// Mitsubishi GX Developer project: PLC_PCO520L2   PLC: Q06UDEH   RS485 Communication_STX

PROGRAM ST340_RS
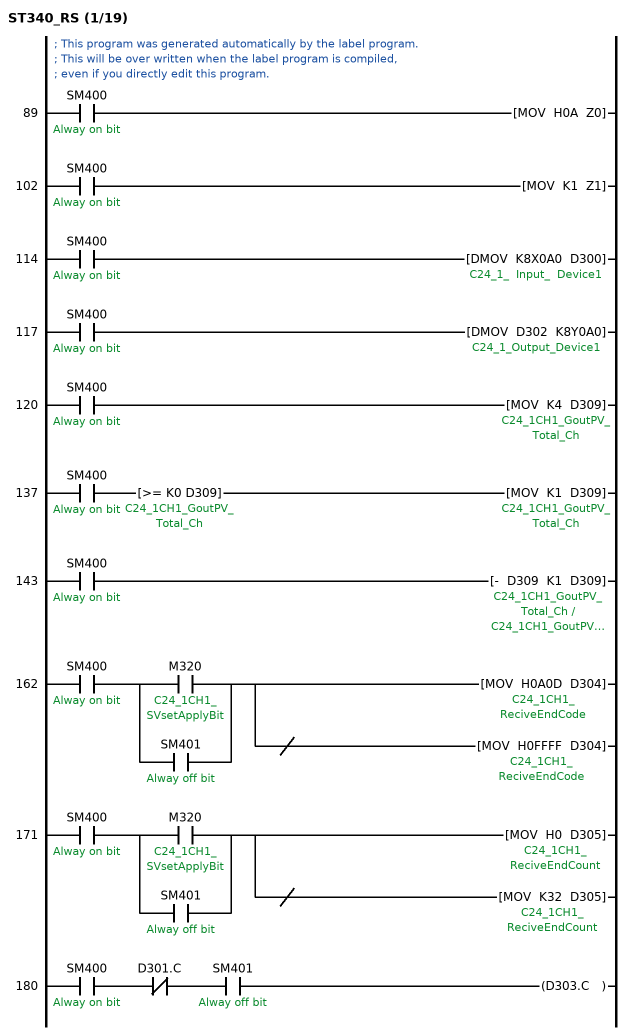
; This program was generated automatically by the label program.
; This will be over written when the label program is compiled,
; even if you directly edit this program.
89    LD      SM400  ; Alway on bit
      MOV     H0A Z0
        [note] Module IO Number
102   LD      SM400  ; Alway on bit
      MOV     K1 Z1
        [note] Channel Number
114   LD      SM400  ; Alway on bit
      DMOV    K8X0A0 D300  ; CH1 Transmission normal completi / C24_1_  Input_  Device1
117   LD      SM400  ; Alway on bit
      DMOV    D302 K8Y0A0  ; C24_1_Output_Device1 / CH1 Transmission request
120   LD      SM400  ; Alway on bit
      MOV     K4 D309  ; C24_1CH1_GoutPV_Total_Ch
        [note] Controller Channel Count
137   LD      SM400  ; Alway on bit
      AND>=   K0 D309  ; C24_1CH1_GoutPV_Total_Ch
      MOV     K1 D309
143   LD      SM400  ; Alway on bit
      -       D309 K1 D309
        [note] Controller Channel Count
162   LD      SM400  ; Alway on bit
      LD      M320  ; C24_1CH1_SVsetApplyBit
      OR      SM401  ; Alway off bit
      ANB
      MOV     H0A0D D304  ; C24_1CH1_ReciveEndCode
      INV
      MOV     H0FFFF D304
171   LD      SM400  ; Alway on bit
      LD      M320  ; C24_1CH1_SVsetApplyBit
      OR      SM401  ; Alway off bit
      ANB
      MOV     H0 D305  ; C24_1CH1_ReciveEndCount
      INV
      MOV     K32 D305
180   LD      SM400  ; Alway on bit
      ANI     D301.C
      AND     SM401  ; Alway off bit
      OUT     D303.C
        [note] System汲沥檬扁拳
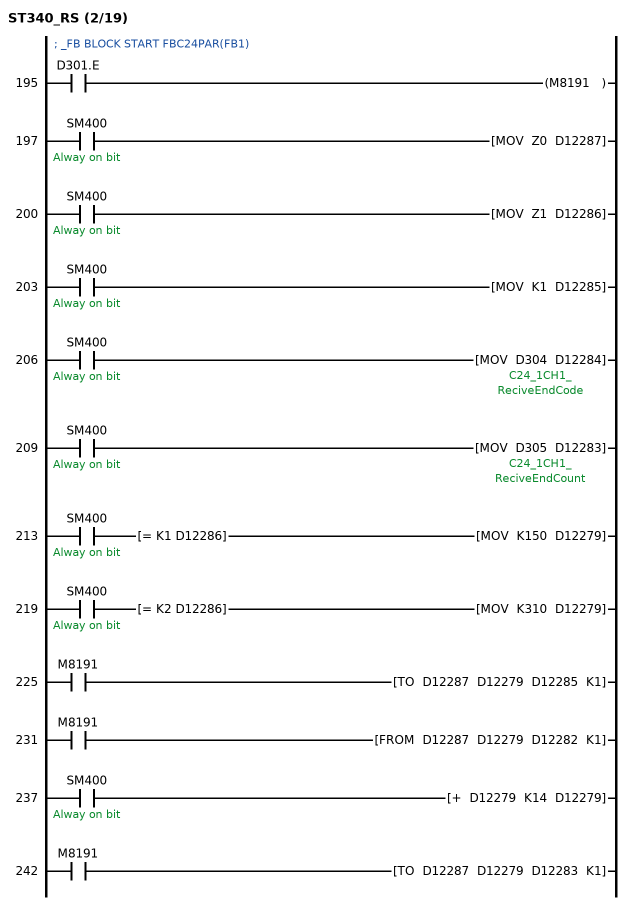
; _FB BLOCK START FBC24PAR(FB1)
195   LD      D301.E
      OUT     M8191
197   LD      SM400  ; Alway on bit
      MOV     Z0 D12287
200   LD      SM400  ; Alway on bit
      MOV     Z1 D12286
203   LD      SM400  ; Alway on bit
      MOV     K1 D12285
206   LD      SM400  ; Alway on bit
      MOV     D304 D12284
209   LD      SM400  ; Alway on bit
      MOV     D305 D12283
; FB START
213   LD      SM400  ; Alway on bit
      AND=    K1 D12286
      MOV     K150 D12279
219   LD      SM400  ; Alway on bit
      AND=    K2 D12286
      MOV     K310 D12279
225   LD      M8191
      TO      D12287 D12279 D12285 K1
231   LD      M8191
      FROM    D12287 D12279 D12282 K1
237   LD      SM400  ; Alway on bit
      +       D12279 K14 D12279
242   LD      M8191
      TO      D12287 D12279 D12283 K1
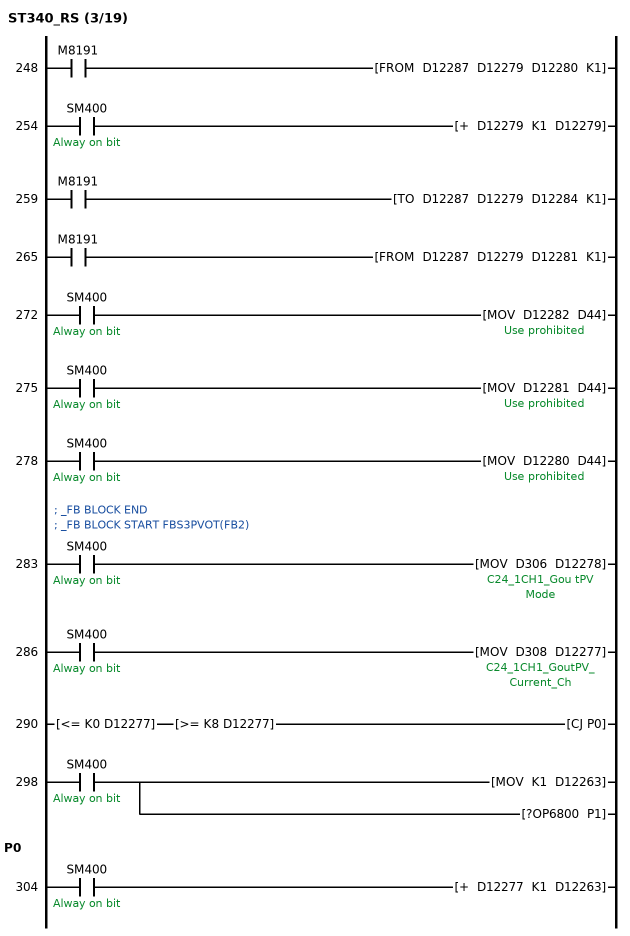
248   LD      M8191
      FROM    D12287 D12279 D12280 K1
254   LD      SM400  ; Alway on bit
      +       D12279 K1 D12279
259   LD      M8191
      TO      D12287 D12279 D12284 K1
265   LD      M8191
      FROM    D12287 D12279 D12281 K1
; FB END
272   LD      SM400  ; Alway on bit
      MOV     D12282 D44  ; Use prohibited
275   LD      SM400  ; Alway on bit
      MOV     D12281 D44
278   LD      SM400  ; Alway on bit
      MOV     D12280 D44
; _FB BLOCK END
; _FB BLOCK START FBS3PVOT(FB2)
283   LD      SM400  ; Alway on bit
      MOV     D306 D12278  ; C24_1CH1_Gou tPV Mode
286   LD      SM400  ; Alway on bit
      MOV     D308 D12277  ; C24_1CH1_GoutPV_Current_Ch
; FB START
290   LD<=    K0 D12277
      AND>=   K8 D12277
      CJ      P0
298   LD      SM400  ; Alway on bit
      MOV     K1 D12263
      ?OP6800 P1
      P0
304   LD      SM400  ; Alway on bit
      +       D12277 K1 D12263
      P1
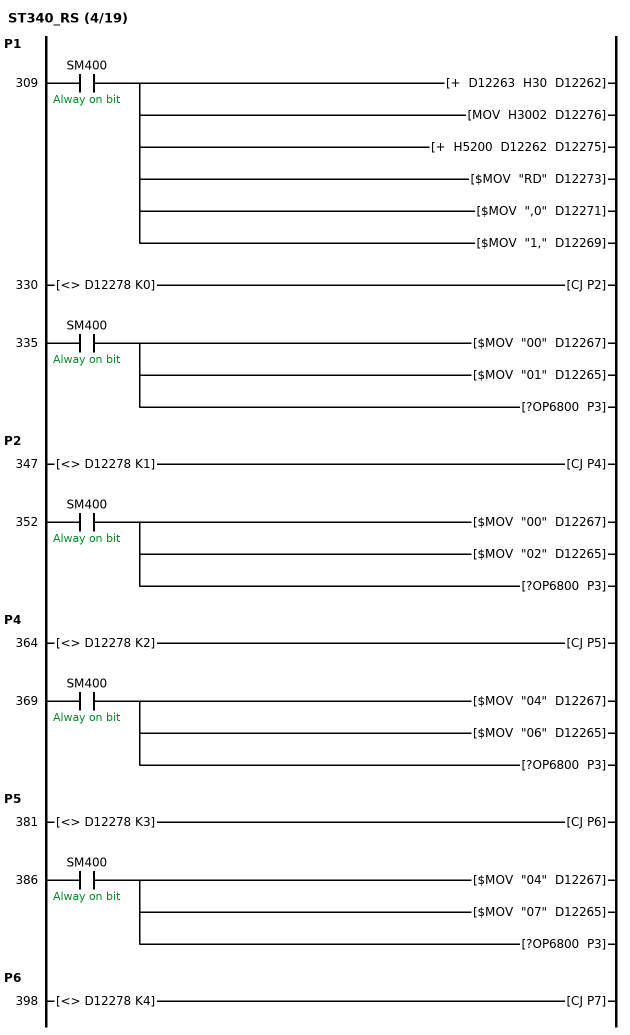
309   LD      SM400  ; Alway on bit
      +       D12263 H30 D12262
      MOV     H3002 D12276
      +       H5200 D12262 D12275
      $MOV    "RD" D12273
      $MOV    ",0" D12271
      $MOV    "1," D12269
330   LD<>    D12278 K0
      CJ      P2
335   LD      SM400  ; Alway on bit
      $MOV    "00" D12267
      $MOV    "01" D12265
      ?OP6800 P3
      P2
347   LD<>    D12278 K1
      CJ      P4
352   LD      SM400  ; Alway on bit
      $MOV    "00" D12267
      $MOV    "02" D12265
      ?OP6800 P3
      P4
364   LD<>    D12278 K2
      CJ      P5
369   LD      SM400  ; Alway on bit
      $MOV    "04" D12267
      $MOV    "06" D12265
      ?OP6800 P3
      P5
381   LD<>    D12278 K3
      CJ      P6
386   LD      SM400  ; Alway on bit
      $MOV    "04" D12267
      $MOV    "07" D12265
      ?OP6800 P3
      P6
398   LD<>    D12278 K4
      CJ      P7
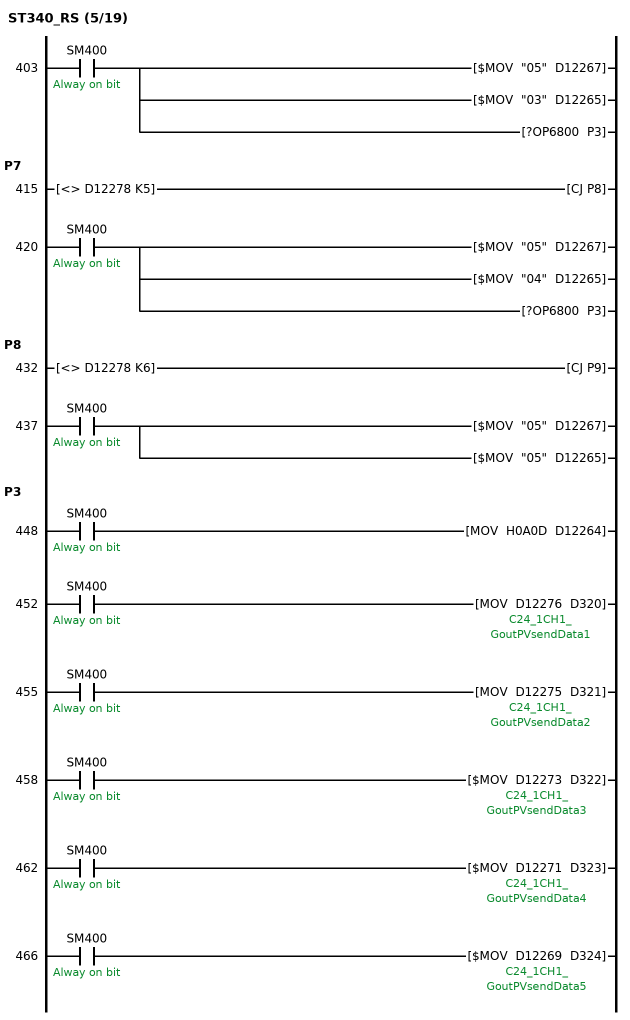
403   LD      SM400  ; Alway on bit
      $MOV    "05" D12267
      $MOV    "03" D12265
      ?OP6800 P3
      P7
415   LD<>    D12278 K5
      CJ      P8
420   LD      SM400  ; Alway on bit
      $MOV    "05" D12267
      $MOV    "04" D12265
      ?OP6800 P3
      P8
432   LD<>    D12278 K6
      CJ      P9
437   LD      SM400  ; Alway on bit
      $MOV    "05" D12267
      $MOV    "05" D12265
      P9
      P3
448   LD      SM400  ; Alway on bit
      MOV     H0A0D D12264
; FB END
452   LD      SM400  ; Alway on bit
      MOV     D12276 D320  ; C24_1CH1_GoutPVsendData1
455   LD      SM400  ; Alway on bit
      MOV     D12275 D321  ; C24_1CH1_GoutPVsendData2
458   LD      SM400  ; Alway on bit
      $MOV    D12273 D322  ; C24_1CH1_GoutPVsendData3
462   LD      SM400  ; Alway on bit
      $MOV    D12271 D323  ; C24_1CH1_GoutPVsendData4
466   LD      SM400  ; Alway on bit
      $MOV    D12269 D324  ; C24_1CH1_GoutPVsendData5
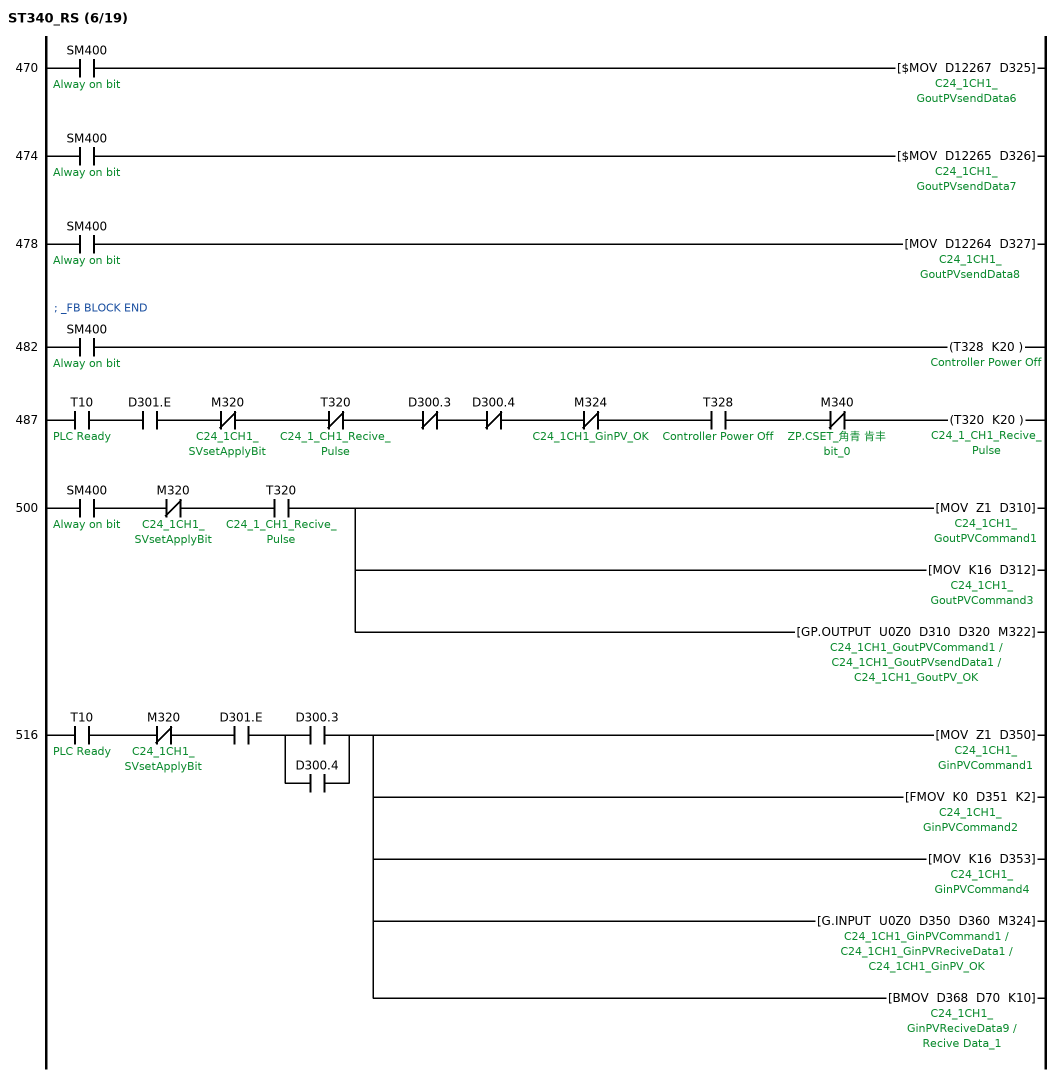
470   LD      SM400  ; Alway on bit
      $MOV    D12267 D325  ; C24_1CH1_GoutPVsendData6
474   LD      SM400  ; Alway on bit
      $MOV    D12265 D326  ; C24_1CH1_GoutPVsendData7
478   LD      SM400  ; Alway on bit
      MOV     D12264 D327  ; C24_1CH1_GoutPVsendData8
; _FB BLOCK END
482   LD      SM400  ; Alway on bit
      OUT     T328 K20  ; Controller Power Off
487   LD      T10  ; PLC Ready
      AND     D301.E
      ANI     M320  ; C24_1CH1_SVsetApplyBit
      ANI     T320  ; C24_1_CH1_Recive_Pulse
      ANI     D300.3
      ANI     D300.4
      ANI     M324  ; C24_1CH1_GinPV_OK
      AND     T328  ; Controller Power Off
      ANI     M340  ; ZP.CSET_角青 肯丰 bit_0
      OUTH    T320 K20  ; C24_1_CH1_Recive_Pulse
500   LD      SM400  ; Alway on bit
      ANI     M320  ; C24_1CH1_SVsetApplyBit
      AND     T320  ; C24_1_CH1_Recive_Pulse
      MOV     Z1 D310  ; C24_1CH1_GoutPVCommand1
      MOV     K16 D312  ; C24_1CH1_GoutPVCommand3
      GP.OUTPUT U0Z0 D310 D320 M322  ; C24_1CH1_GoutPV_OK
516   LD      T10  ; PLC Ready
      ANI     M320  ; C24_1CH1_SVsetApplyBit
      AND     D301.E
      LD      D300.3
      OR      D300.4
      ANB
      MOV     Z1 D350  ; C24_1CH1_GinPVCommand1
      FMOV    K0 D351 K2  ; C24_1CH1_GinPVCommand2
      MOV     K16 D353  ; C24_1CH1_GinPVCommand4
      G.INPUT U0Z0 D350 D360 M324  ; C24_1CH1_GinPVReciveData1
      BMOV    D368 D70 K10  ; C24_1CH1_GinPVReciveData9 / Recive Data_1
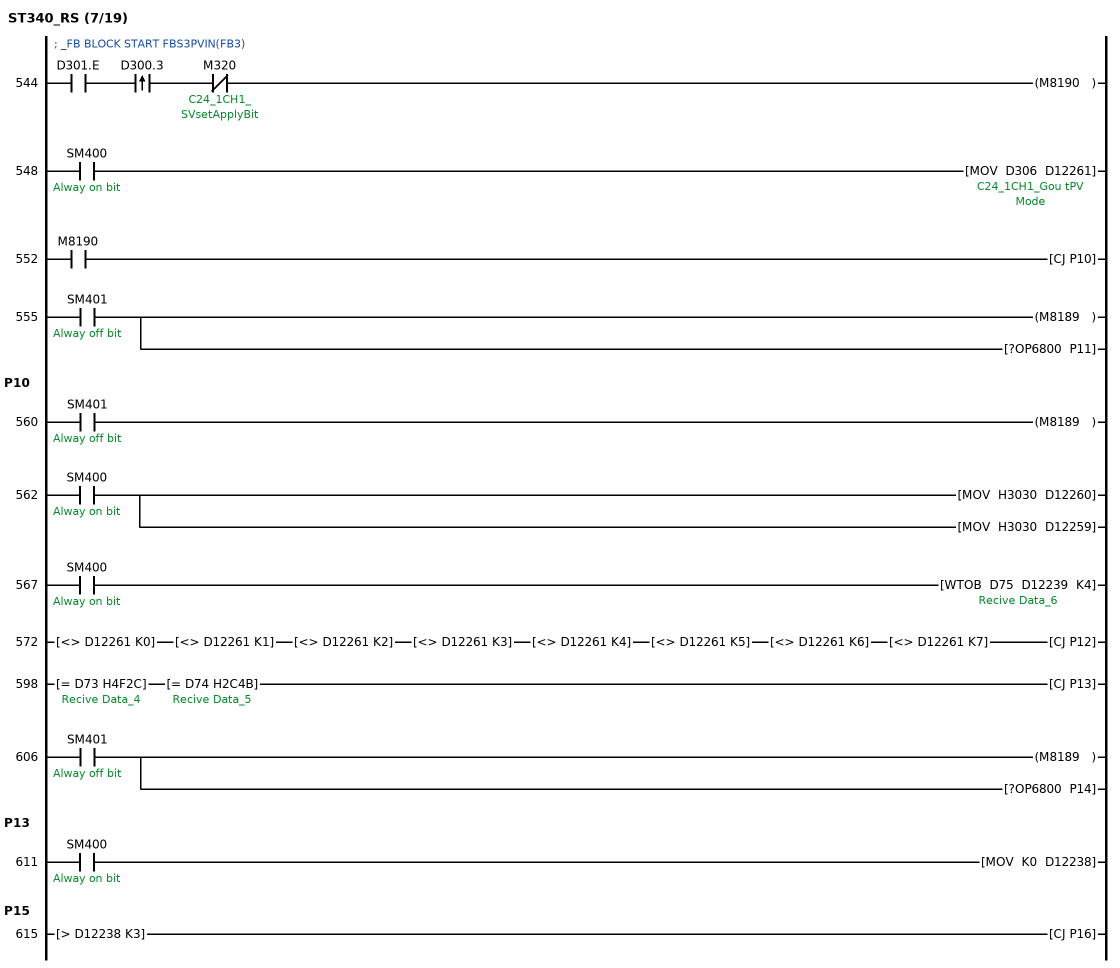
; _FB BLOCK START FBS3PVIN(FB3)
544   LD      D301.E
      ANDP    D300.3
      ANI     M320  ; C24_1CH1_SVsetApplyBit
      OUT     M8190
548   LD      SM400  ; Alway on bit
      MOV     D306 D12261
; FB START
552   LD      M8190
      CJ      P10
555   LD      SM401  ; Alway off bit
      OUT     M8189
      ?OP6800 P11
      P10
560   LD      SM401  ; Alway off bit
      OUT     M8189
562   LD      SM400  ; Alway on bit
      MOV     H3030 D12260
      MOV     H3030 D12259
567   LD      SM400  ; Alway on bit
      WTOB    D75 D12239 K4  ; Recive Data_6
572   LD<>    D12261 K0
      AND<>   D12261 K1
      AND<>   D12261 K2
      AND<>   D12261 K3
      AND<>   D12261 K4
      AND<>   D12261 K5
      AND<>   D12261 K6
      AND<>   D12261 K7
      CJ      P12
598   LD=     D73 H4F2C  ; Recive Data_4
      AND=    D74 H2C4B  ; Recive Data_5
      CJ      P13
606   LD      SM401  ; Alway off bit
      OUT     M8189
      ?OP6800 P14
      P13
611   LD      SM400  ; Alway on bit
      MOV     K0 D12238
      P15
615   LD>     D12238 K3
      CJ      P16
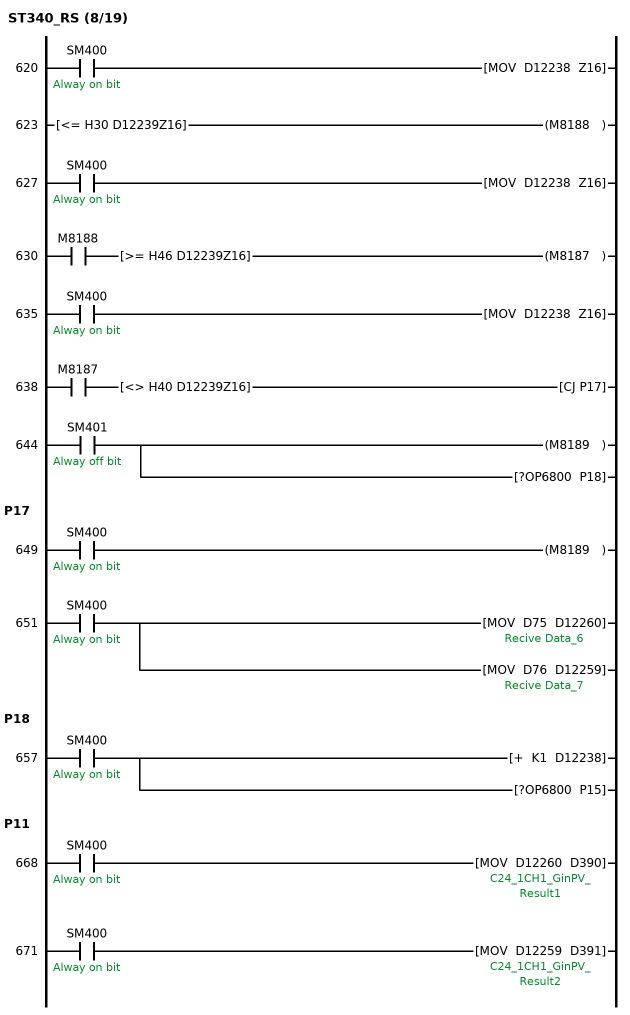
620   LD      SM400  ; Alway on bit
      MOV     D12238 Z16
623   LD<=    H30 D12239Z16
      OUT     M8188
627   LD      SM400  ; Alway on bit
      MOV     D12238 Z16
630   LD      M8188
      AND>=   H46 D12239Z16
      OUT     M8187
635   LD      SM400  ; Alway on bit
      MOV     D12238 Z16
638   LD      M8187
      AND<>   H40 D12239Z16
      CJ      P17
644   LD      SM401  ; Alway off bit
      OUT     M8189
      ?OP6800 P18
      P17
649   LD      SM400  ; Alway on bit
      OUT     M8189
651   LD      SM400  ; Alway on bit
      MOV     D75 D12260
      MOV     D76 D12259  ; Recive Data_7
      P18
657   LD      SM400  ; Alway on bit
      +       K1 D12238
      ?OP6800 P15
      P16
      P14
      P12
      P11
; FB END
668   LD      SM400  ; Alway on bit
      MOV     D12260 D390  ; C24_1CH1_GinPV_Result1
671   LD      SM400  ; Alway on bit
      MOV     D12259 D391  ; C24_1CH1_GinPV_Result2
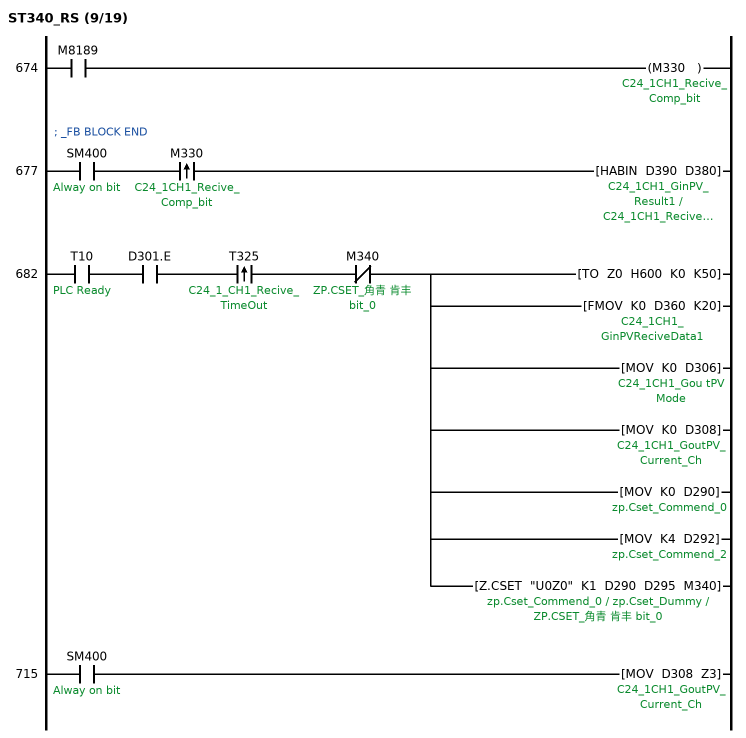
674   LD      M8189
      OUT     M330  ; C24_1CH1_Recive_Comp_bit
; _FB BLOCK END
677   LD      SM400  ; Alway on bit
      ANDP    M330  ; C24_1CH1_Recive_Comp_bit
      HABIN   D390 D380  ; C24_1CH1_Recive_Value_1
682   LD      T10  ; PLC Ready
      AND     D301.E
      ANDP    T325  ; C24_1_CH1_Recive_TimeOut
      ANI     M340  ; ZP.CSET_角青 肯丰 bit_0
      TO      Z0 H600 K0 K50
      FMOV    K0 D360 K20
      MOV     K0 D306
      MOV     K0 D308
      MOV     K0 D290  ; zp.Cset_Commend_0
      MOV     K4 D292  ; zp.Cset_Commend_2
      Z.CSET  "U0Z0" K1 D290 D295 M340  ; zp.Cset_Dummy
715   LD      SM400  ; Alway on bit
      MOV     D308 Z3
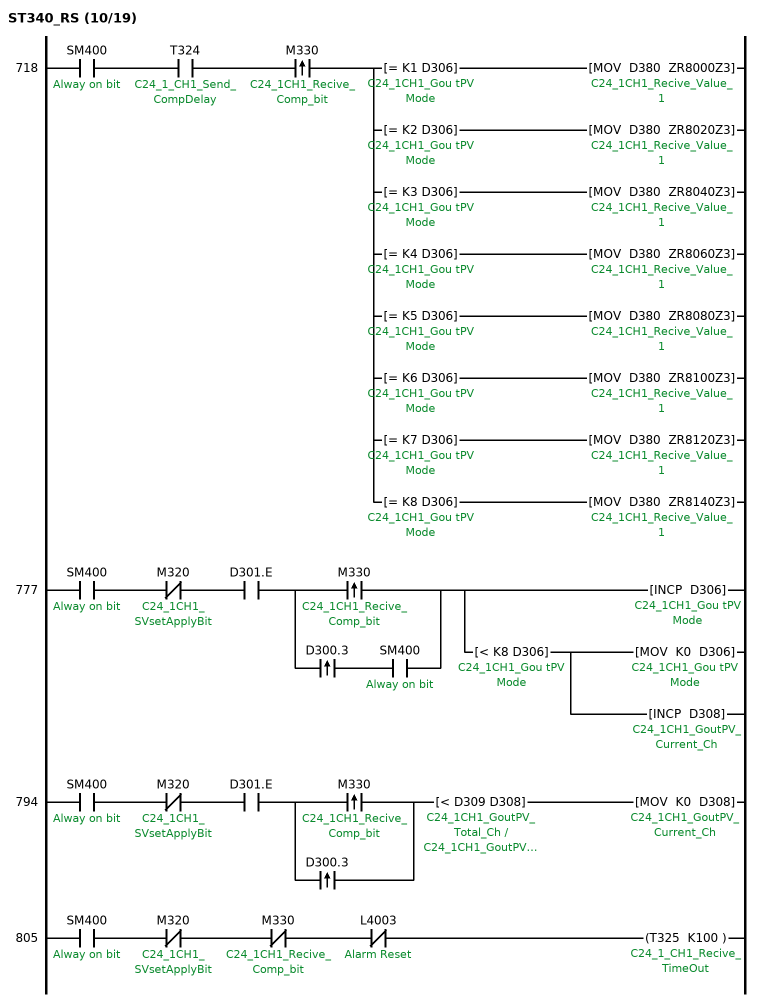
718   LD      SM400  ; Alway on bit
      AND     T324  ; C24_1_CH1_Send_CompDelay
      ANDP    M330  ; C24_1CH1_Recive_Comp_bit
      MPS
      AND=    K1 D306  ; C24_1CH1_Gou tPV Mode
      MOV     D380 ZR8000Z3
      MRD
      AND=    K2 D306  ; C24_1CH1_Gou tPV Mode
      MOV     D380 ZR8020Z3
      MRD
      AND=    K3 D306  ; C24_1CH1_Gou tPV Mode
      MOV     D380 ZR8040Z3
      MRD
      AND=    K4 D306  ; C24_1CH1_Gou tPV Mode
      MOV     D380 ZR8060Z3
      MRD
      AND=    K5 D306  ; C24_1CH1_Gou tPV Mode
      MOV     D380 ZR8080Z3
      MRD
      AND=    K6 D306  ; C24_1CH1_Gou tPV Mode
      MOV     D380 ZR8100Z3
      MRD
      AND=    K7 D306  ; C24_1CH1_Gou tPV Mode
      MOV     D380 ZR8120Z3
      MPP
      AND=    K8 D306  ; C24_1CH1_Gou tPV Mode
      MOV     D380 ZR8140Z3
777   LD      SM400  ; Alway on bit
      ANI     M320  ; C24_1CH1_SVsetApplyBit
      AND     D301.E
      LDP     M330  ; C24_1CH1_Recive_Comp_bit
      LDP     D300.3
      AND     SM400  ; Alway on bit
      ORB
      ANB
      INCP    D306
      AND<    K8 D306  ; C24_1CH1_Gou tPV Mode
      MOV     K0 D306
      INCP    D308
794   LD      SM400  ; Alway on bit
      ANI     M320  ; C24_1CH1_SVsetApplyBit
      AND     D301.E
      LDP     M330  ; C24_1CH1_Recive_Comp_bit
      ORP     D300.3
      ANB
      AND<    D309 D308  ; C24_1CH1_GoutPV_Total_Ch / C24_1CH1_GoutPV_Current_Ch
      MOV     K0 D308
805   LD      SM400  ; Alway on bit
      ANI     M320  ; C24_1CH1_SVsetApplyBit
      ANI     M330  ; C24_1CH1_Recive_Comp_bit
      ANI     L4003  ; Alarm Reset
      OUT     T325 K100  ; C24_1_CH1_Recive_TimeOut
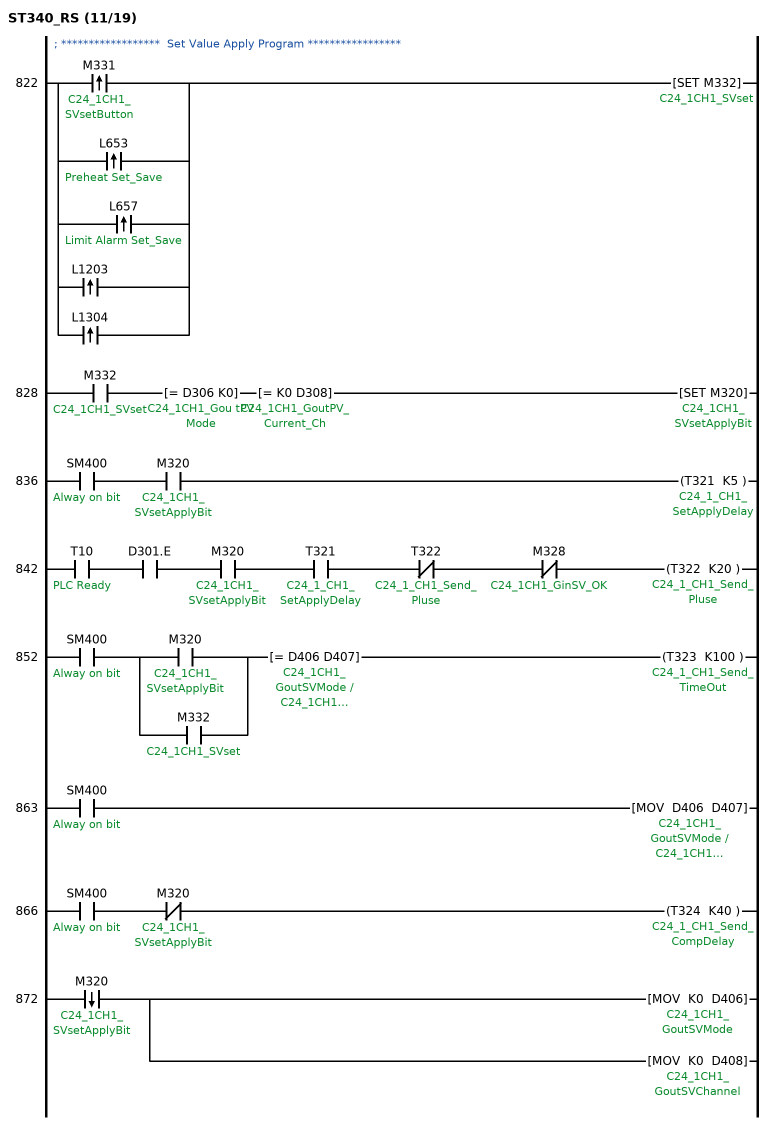
; 
; 
; 
; 
; ******************  Set Value Apply Program *****************
822   LDP     M331  ; C24_1CH1_SVsetButton
      ORP     L653  ; Preheat Set_Save
      ORP     L657  ; Limit Alarm Set_Save
      ORP     L1203
      ORP     L1304
      SET     M332  ; C24_1CH1_SVset
828   LD      M332  ; C24_1CH1_SVset
      AND=    D306 K0  ; C24_1CH1_Gou tPV Mode
      AND=    K0 D308  ; C24_1CH1_GoutPV_Current_Ch
      SET     M320  ; C24_1CH1_SVsetApplyBit
836   LD      SM400  ; Alway on bit
      AND     M320  ; C24_1CH1_SVsetApplyBit
      OUT     T321 K5  ; C24_1_CH1_SetApplyDelay
842   LD      T10  ; PLC Ready
      AND     D301.E
      AND     M320  ; C24_1CH1_SVsetApplyBit
      AND     T321  ; C24_1_CH1_SetApplyDelay
      ANI     T322  ; C24_1_CH1_Send_Pluse
      ANI     M328  ; C24_1CH1_GinSV_OK
      OUTH    T322 K20  ; C24_1_CH1_Send_Pluse
852   LD      SM400  ; Alway on bit
      LD      M320  ; C24_1CH1_SVsetApplyBit
      OR      M332  ; C24_1CH1_SVset
      ANB
      AND=    D406 D407  ; C24_1CH1_GoutSVMode / C24_1CH1_GoutSVModeBuffer
      OUT     T323 K100  ; C24_1_CH1_Send_TimeOut
863   LD      SM400  ; Alway on bit
      MOV     D406 D407
866   LD      SM400  ; Alway on bit
      ANI     M320  ; C24_1CH1_SVsetApplyBit
      OUTH    T324 K40  ; C24_1_CH1_Send_CompDelay
872   LDF     M320  ; C24_1CH1_SVsetApplyBit
      MOV     K0 D406
      MOV     K0 D408  ; C24_1CH1_GoutSVChannel
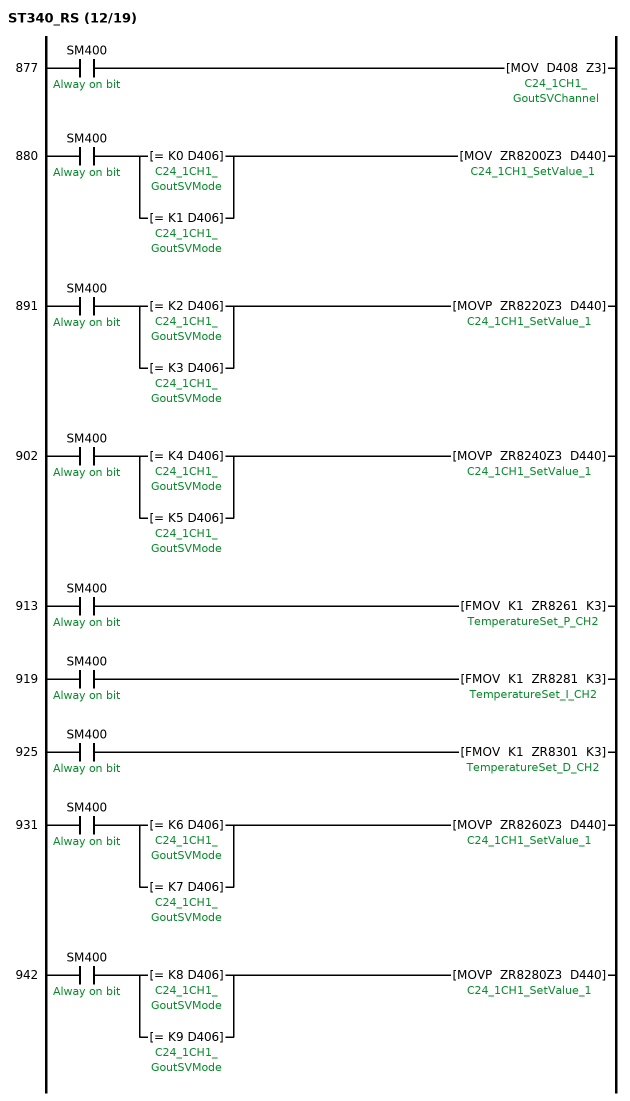
877   LD      SM400  ; Alway on bit
      MOV     D408 Z3
880   LD      SM400  ; Alway on bit
      LD=     K0 D406  ; C24_1CH1_GoutSVMode
      OR=     K1 D406  ; C24_1CH1_GoutSVMode
      ANB
      MOV     ZR8200Z3 D440  ; C24_1CH1_SetValue_1
891   LD      SM400  ; Alway on bit
      LD=     K2 D406  ; C24_1CH1_GoutSVMode
      OR=     K3 D406  ; C24_1CH1_GoutSVMode
      ANB
      MOVP    ZR8220Z3 D440
902   LD      SM400  ; Alway on bit
      LD=     K4 D406  ; C24_1CH1_GoutSVMode
      OR=     K5 D406  ; C24_1CH1_GoutSVMode
      ANB
      MOVP    ZR8240Z3 D440
913   LD      SM400  ; Alway on bit
      FMOV    K1 ZR8261 K3  ; TemperatureSet_P_CH2
919   LD      SM400  ; Alway on bit
      FMOV    K1 ZR8281 K3  ; TemperatureSet_I_CH2
925   LD      SM400  ; Alway on bit
      FMOV    K1 ZR8301 K3  ; TemperatureSet_D_CH2
931   LD      SM400  ; Alway on bit
      LD=     K6 D406  ; C24_1CH1_GoutSVMode
      OR=     K7 D406  ; C24_1CH1_GoutSVMode
      ANB
      MOVP    ZR8260Z3 D440
942   LD      SM400  ; Alway on bit
      LD=     K8 D406  ; C24_1CH1_GoutSVMode
      OR=     K9 D406  ; C24_1CH1_GoutSVMode
      ANB
      MOVP    ZR8280Z3 D440
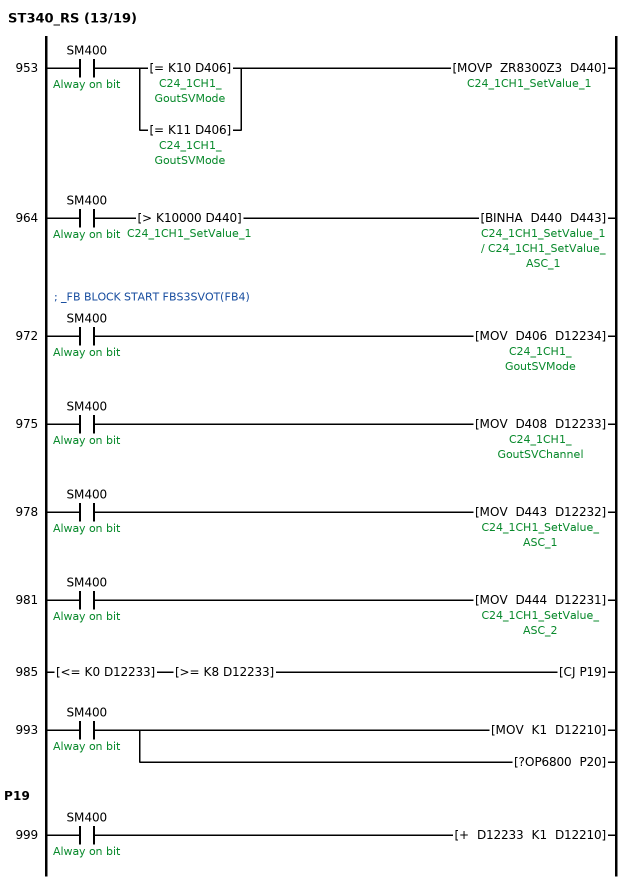
953   LD      SM400  ; Alway on bit
      LD=     K10 D406  ; C24_1CH1_GoutSVMode
      OR=     K11 D406  ; C24_1CH1_GoutSVMode
      ANB
      MOVP    ZR8300Z3 D440
964   LD      SM400  ; Alway on bit
      AND>    K10000 D440  ; C24_1CH1_SetValue_1
      BINHA   D440 D443  ; C24_1CH1_SetValue_ASC_1
; _FB BLOCK START FBS3SVOT(FB4)
972   LD      SM400  ; Alway on bit
      MOV     D406 D12234
975   LD      SM400  ; Alway on bit
      MOV     D408 D12233
978   LD      SM400  ; Alway on bit
      MOV     D443 D12232
981   LD      SM400  ; Alway on bit
      MOV     D444 D12231  ; C24_1CH1_SetValue_ASC_2
; FB START
985   LD<=    K0 D12233
      AND>=   K8 D12233
      CJ      P19
993   LD      SM400  ; Alway on bit
      MOV     K1 D12210
      ?OP6800 P20
      P19
999   LD      SM400  ; Alway on bit
      +       D12233 K1 D12210
      P20
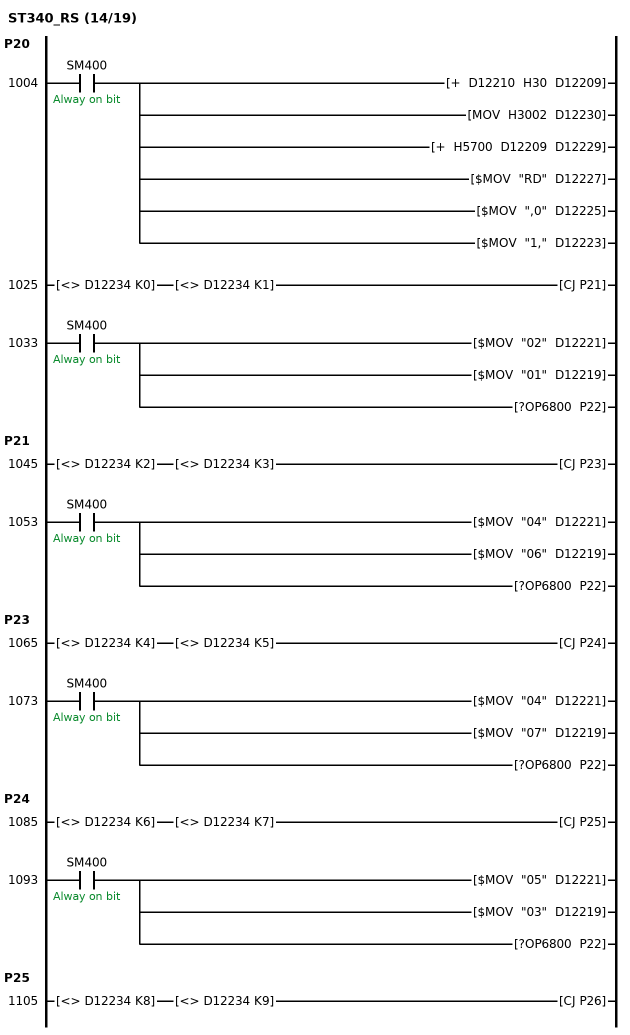
1004  LD      SM400  ; Alway on bit
      +       D12210 H30 D12209
      MOV     H3002 D12230
      +       H5700 D12209 D12229
      $MOV    "RD" D12227
      $MOV    ",0" D12225
      $MOV    "1," D12223
1025  LD<>    D12234 K0
      AND<>   D12234 K1
      CJ      P21
1033  LD      SM400  ; Alway on bit
      $MOV    "02" D12221
      $MOV    "01" D12219
      ?OP6800 P22
      P21
1045  LD<>    D12234 K2
      AND<>   D12234 K3
      CJ      P23
1053  LD      SM400  ; Alway on bit
      $MOV    "04" D12221
      $MOV    "06" D12219
      ?OP6800 P22
      P23
1065  LD<>    D12234 K4
      AND<>   D12234 K5
      CJ      P24
1073  LD      SM400  ; Alway on bit
      $MOV    "04" D12221
      $MOV    "07" D12219
      ?OP6800 P22
      P24
1085  LD<>    D12234 K6
      AND<>   D12234 K7
      CJ      P25
1093  LD      SM400  ; Alway on bit
      $MOV    "05" D12221
      $MOV    "03" D12219
      ?OP6800 P22
      P25
1105  LD<>    D12234 K8
      AND<>   D12234 K9
      CJ      P26
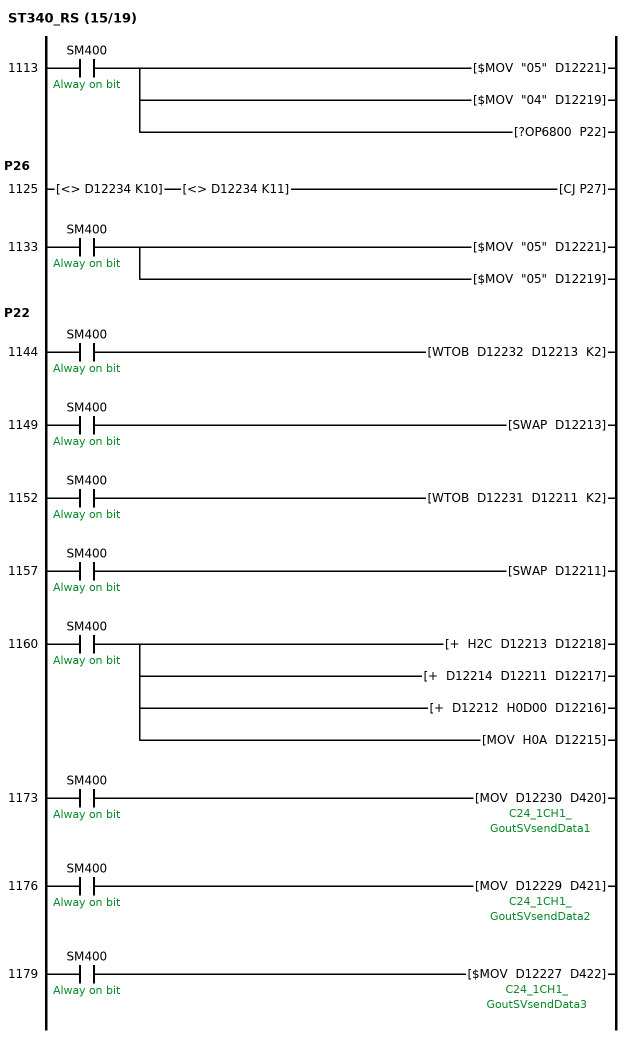
1113  LD      SM400  ; Alway on bit
      $MOV    "05" D12221
      $MOV    "04" D12219
      ?OP6800 P22
      P26
1125  LD<>    D12234 K10
      AND<>   D12234 K11
      CJ      P27
1133  LD      SM400  ; Alway on bit
      $MOV    "05" D12221
      $MOV    "05" D12219
      P27
      P22
1144  LD      SM400  ; Alway on bit
      WTOB    D12232 D12213 K2
1149  LD      SM400  ; Alway on bit
      SWAP    D12213
1152  LD      SM400  ; Alway on bit
      WTOB    D12231 D12211 K2
1157  LD      SM400  ; Alway on bit
      SWAP    D12211
1160  LD      SM400  ; Alway on bit
      +       H2C D12213 D12218
      +       D12214 D12211 D12217
      +       D12212 H0D00 D12216
      MOV     H0A D12215
; FB END
1173  LD      SM400  ; Alway on bit
      MOV     D12230 D420  ; C24_1CH1_GoutSVsendData1
1176  LD      SM400  ; Alway on bit
      MOV     D12229 D421  ; C24_1CH1_GoutSVsendData2
1179  LD      SM400  ; Alway on bit
      $MOV    D12227 D422  ; C24_1CH1_GoutSVsendData3
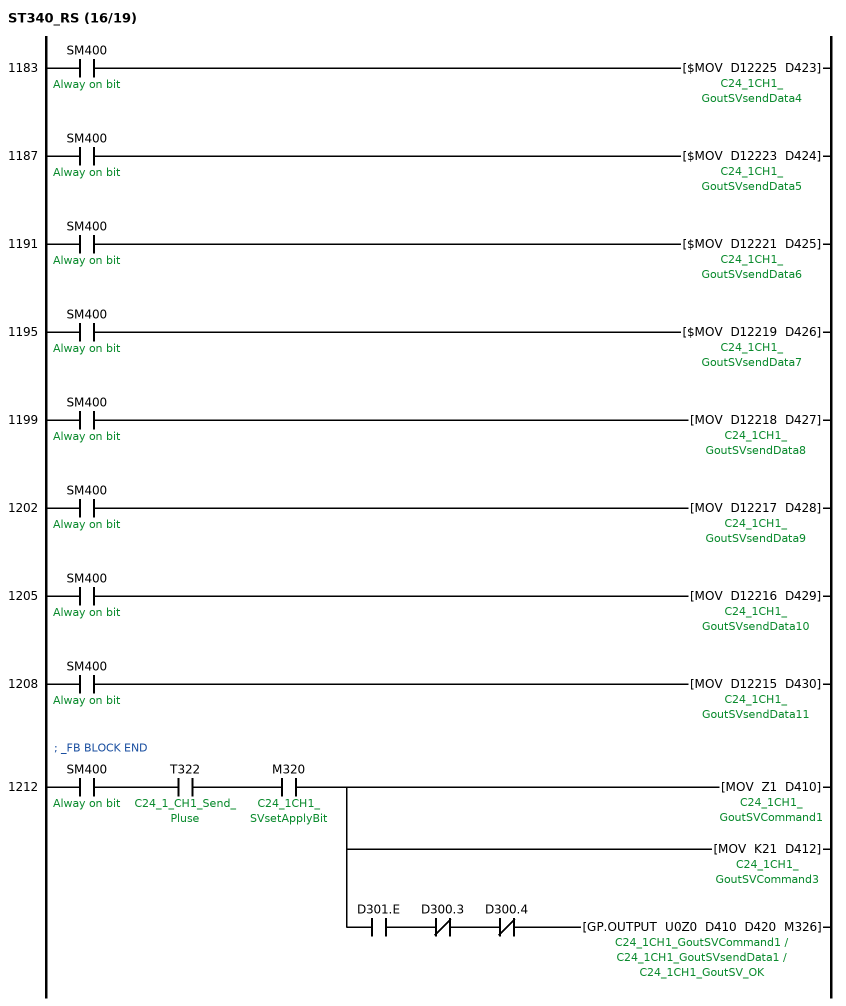
1183  LD      SM400  ; Alway on bit
      $MOV    D12225 D423  ; C24_1CH1_GoutSVsendData4
1187  LD      SM400  ; Alway on bit
      $MOV    D12223 D424  ; C24_1CH1_GoutSVsendData5
1191  LD      SM400  ; Alway on bit
      $MOV    D12221 D425  ; C24_1CH1_GoutSVsendData6
1195  LD      SM400  ; Alway on bit
      $MOV    D12219 D426  ; C24_1CH1_GoutSVsendData7
1199  LD      SM400  ; Alway on bit
      MOV     D12218 D427  ; C24_1CH1_GoutSVsendData8
1202  LD      SM400  ; Alway on bit
      MOV     D12217 D428  ; C24_1CH1_GoutSVsendData9
1205  LD      SM400  ; Alway on bit
      MOV     D12216 D429  ; C24_1CH1_GoutSVsendData10
1208  LD      SM400  ; Alway on bit
      MOV     D12215 D430  ; C24_1CH1_GoutSVsendData11
; _FB BLOCK END
1212  LD      SM400  ; Alway on bit
      AND     T322  ; C24_1_CH1_Send_Pluse
      AND     M320  ; C24_1CH1_SVsetApplyBit
      MOV     Z1 D410  ; C24_1CH1_GoutSVCommand1
      MOV     K21 D412  ; C24_1CH1_GoutSVCommand3
      AND     D301.E
      ANI     D300.3
      ANI     D300.4
      GP.OUTPUT U0Z0 D410 D420 M326  ; C24_1CH1_GoutSV_OK
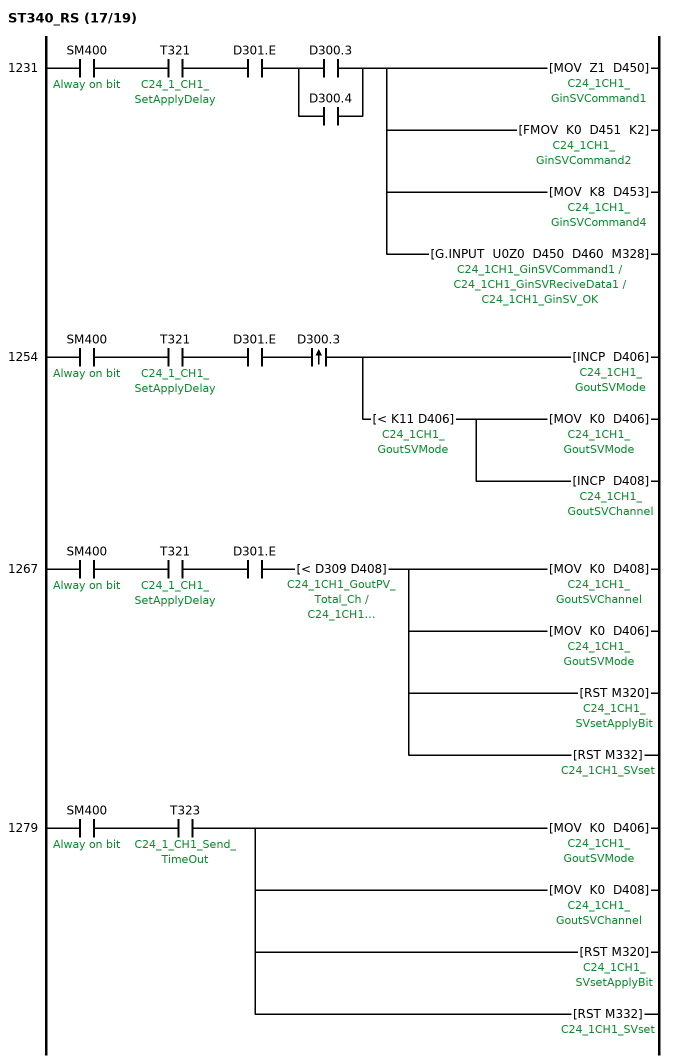
1231  LD      SM400  ; Alway on bit
      AND     T321  ; C24_1_CH1_SetApplyDelay
      AND     D301.E
      LD      D300.3
      OR      D300.4
      ANB
      MOV     Z1 D450  ; C24_1CH1_GinSVCommand1
      FMOV    K0 D451 K2  ; C24_1CH1_GinSVCommand2
      MOV     K8 D453  ; C24_1CH1_GinSVCommand4
      G.INPUT U0Z0 D450 D460 M328  ; C24_1CH1_GinSVReciveData1
1254  LD      SM400  ; Alway on bit
      AND     T321  ; C24_1_CH1_SetApplyDelay
      AND     D301.E
      ANDP    D300.3
      INCP    D406
      AND<    K11 D406  ; C24_1CH1_GoutSVMode
      MOV     K0 D406
      INCP    D408
1267  LD      SM400  ; Alway on bit
      AND     T321  ; C24_1_CH1_SetApplyDelay
      AND     D301.E
      AND<    D309 D408  ; C24_1CH1_GoutPV_Total_Ch / C24_1CH1_GoutSVChannel
      MOV     K0 D408
      MOV     K0 D406
      RST     M320  ; C24_1CH1_SVsetApplyBit
      RST     M332  ; C24_1CH1_SVset
1279  LD      SM400  ; Alway on bit
      AND     T323  ; C24_1_CH1_Send_TimeOut
      MOV     K0 D406
      MOV     K0 D408
      RST     M320  ; C24_1CH1_SVsetApplyBit
      RST     M332  ; C24_1CH1_SVset
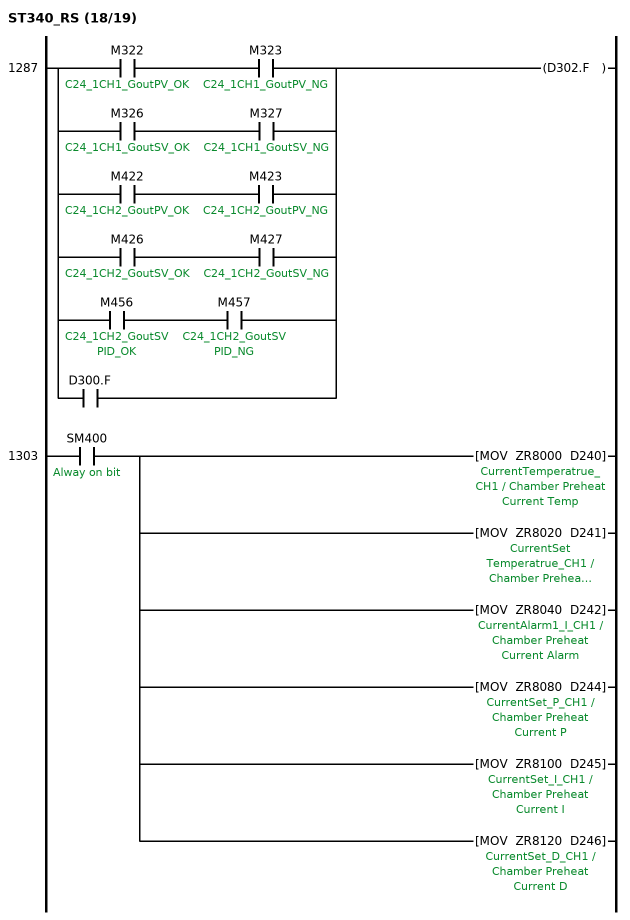
1287  LD      M322  ; C24_1CH1_GoutPV_OK
      AND     M323  ; C24_1CH1_GoutPV_NG
      LD      M326  ; C24_1CH1_GoutSV_OK
      AND     M327  ; C24_1CH1_GoutSV_NG
      ORB
      LD      M422  ; C24_1CH2_GoutPV_OK
      AND     M423  ; C24_1CH2_GoutPV_NG
      ORB
      LD      M426  ; C24_1CH2_GoutSV_OK
      AND     M427  ; C24_1CH2_GoutSV_NG
      ORB
      LD      M456  ; C24_1CH2_GoutSV PID_OK
      AND     M457  ; C24_1CH2_GoutSV PID_NG
      ORB
      OR      D300.F
      OUT     D302.F
1303  LD      SM400  ; Alway on bit
      MOV     ZR8000 D240  ; CurrentTemperatrue_CH1 / Chamber Preheat Current Temp
      MOV     ZR8020 D241  ; CurrentSetTemperatrue_CH1 / Chamber Preheat Current SV Temp
      MOV     ZR8040 D242  ; CurrentAlarm1_I_CH1 / Chamber Preheat Current Alarm
      MOV     ZR8080 D244  ; CurrentSet_P_CH1 / Chamber Preheat Current P
      MOV     ZR8100 D245  ; CurrentSet_I_CH1 / Chamber Preheat Current I
      MOV     ZR8120 D246  ; CurrentSet_D_CH1 / Chamber Preheat Current D
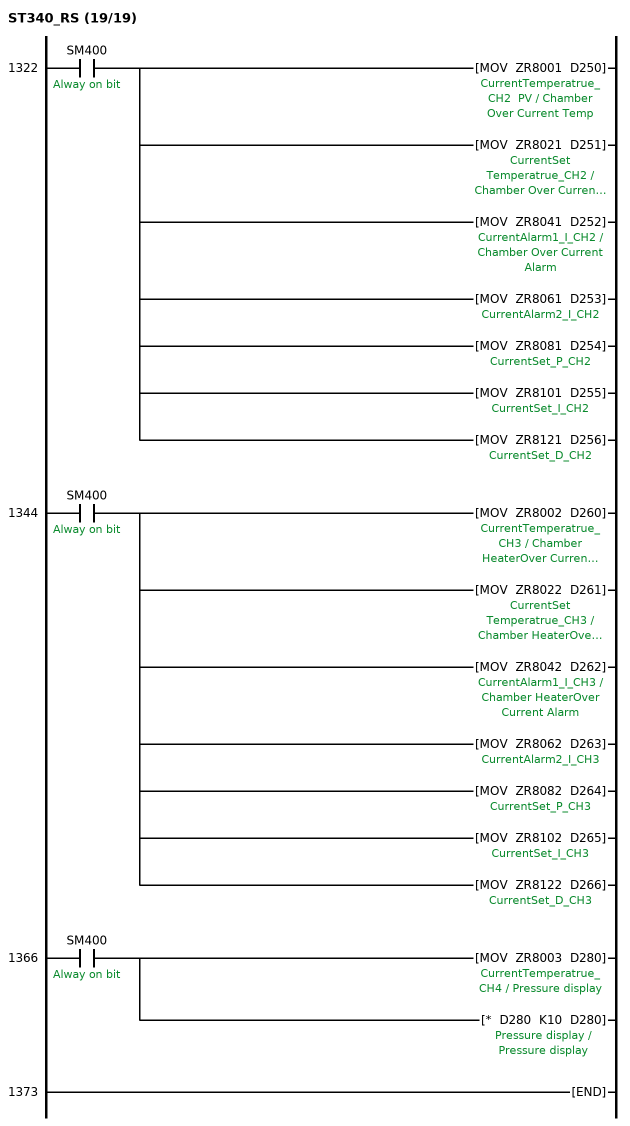
1322  LD      SM400  ; Alway on bit
      MOV     ZR8001 D250  ; CurrentTemperatrue_CH2  PV / Chamber Over Current Temp
      MOV     ZR8021 D251  ; CurrentSetTemperatrue_CH2 / Chamber Over Current SV
      MOV     ZR8041 D252  ; CurrentAlarm1_I_CH2 / Chamber Over Current Alarm
      MOV     ZR8061 D253  ; CurrentAlarm2_I_CH2
      MOV     ZR8081 D254  ; CurrentSet_P_CH2
      MOV     ZR8101 D255  ; CurrentSet_I_CH2
      MOV     ZR8121 D256  ; CurrentSet_D_CH2
1344  LD      SM400  ; Alway on bit
      MOV     ZR8002 D260  ; CurrentTemperatrue_CH3 / Chamber HeaterOver Current Temp
      MOV     ZR8022 D261  ; CurrentSetTemperatrue_CH3 / Chamber HeaterOver Current SV
      MOV     ZR8042 D262  ; CurrentAlarm1_I_CH3 / Chamber HeaterOver Current Alarm
      MOV     ZR8062 D263  ; CurrentAlarm2_I_CH3
      MOV     ZR8082 D264  ; CurrentSet_P_CH3
      MOV     ZR8102 D265  ; CurrentSet_I_CH3
      MOV     ZR8122 D266  ; CurrentSet_D_CH3
1366  LD      SM400  ; Alway on bit
      MOV     ZR8003 D280  ; CurrentTemperatrue_CH4 / Pressure display
      *       D280 K10 D280
1373  END
END_PROGRAM
